// TwinCAT 3 PLC project plc01
// ProgramVersion: 3.1.4026.19
// libraries:
//   Tc2_Standard, * (Beckhoff Automation GmbH)
//   Tc2_System, * (Beckhoff Automation GmbH)
//   Tc2_Utilities, * (Beckhoff Automation GmbH)
//   Tc3_Event, * (www.peterzerlauth.com)
// project tree:
//   / FastTask.TcTTO (not stored), PlcTask.TcTTO (not stored)
//   POUs/ FAST.TcPOU, FB_TestSlow.TcPOU, FB_TestFast.TcPOU, FB_Test1000.TcPOU, MAIN.TcPOU
// real-time tasks:
//   TASK SlowTask: cycle T#20ms, priority 20, ADS port 350
//   TASK FastTask: cycle T#1ms, priority 1, ADS port 351

// ---- POUs/FAST.TcPOU
PROGRAM FAST
VAR
	fbTest:			FB_TestFast;
  	exception:			__SYSTEM.ExceptionCode;	
END_VAR

__TRY
	IF exception = __SYSTEM.ExceptionCode.RTSEXCPT_NOEXCEPTION THEN
// 		fbTest.P_Event.P_Logger:= MAIN.fbLogger;
	
	fbTest();
	
		
	END_IF


__CATCH(exception)


__ENDTRY

END_PROGRAM

// ---- POUs/FB_TestFast.TcPOU
FUNCTION_BLOCK FB_TestFast
VAR_INPUT
END_VAR
VAR_OUTPUT
END_VAR
VAR
	fbEvent: 			Tc3_Event.FB_Event;
	bVerbose:			BOOL;
	bInfo:				BOOL;
	bWarning:			BOOL;
	bError:				BOOL;
	bCritical:			BOOL;

END_VAR

fbEvent();

// Demonstration of FB_Event usage with various log levels and argument types

IF bVerbose THEN
	fbEvent.P_Argument.M_AddINT(134052566194980000);
	fbEvent.P_Argument.M_AddSTRING('mm');
	fbEvent.M_Verbose('V message %s %s');
END_IF

IF bInfo THEN
	fbEvent.P_Argument.M_AddREAL(33.134581234, 3);
	fbEvent.P_Argument.M_AddSTRING('mm');
	fbEvent.M_Info(828536003, 'I message %s %s');
END_IF

IF bWarning THEN
	fbEvent.M_Warning(475719253, 'W message');
	fbEvent.M_Warning(475719253, 'W message');
END_IF

IF bError THEN
	fbEvent.M_Error(475719235, 'E message');
END_IF

IF bCritical THEN
	fbEvent.M_Critical(475719233, 'C message'); ///839384782
END_IF

PROPERTY PUBLIC P_Event : reference to FB_event
GET
P_Event ref= fbEvent;
END_GET
END_PROPERTY

END_FUNCTION_BLOCK

// ---- POUs/FB_TestSlow.TcPOU
FUNCTION_BLOCK FB_TestSlow
VAR_INPUT
END_VAR
VAR_OUTPUT
END_VAR
VAR
	fbEvent: 			Tc3_Event.FB_Event;
	bVerbose:			BOOL;
	bInfo:				BOOL;
	bWarning:			BOOL;
	bError:				BOOL;
	bCritical:			BOOL;

END_VAR

fbEvent();

// Demonstration of FB_Event usage with various log levels and argument types

IF bVerbose THEN
	fbEvent.P_Argument.M_AddINT(134052566194980000);
	fbEvent.P_Argument.M_AddSTRING('mm');
	fbEvent.M_Verbose('V message %s %s');
END_IF

IF bInfo THEN
	fbEvent.P_Argument.M_AddREAL(33.134581234, 3);
	fbEvent.P_Argument.M_AddSTRING('mm');
	fbEvent.M_Info(828536003, 'I message %s %s');
END_IF

IF bWarning THEN
	fbEvent.M_Warning(475719253, 'W message');
	fbEvent.M_Warning(475719253, 'W message');
END_IF

IF bError THEN
	fbEvent.M_Error(475719235, 'E message');
END_IF

IF bCritical THEN
	fbEvent.M_Critical(475719233, 'C message'); ///839384782
	fbEvent.M_Error(849363082, 'Input %s is simulated');
END_IF

PROPERTY PUBLIC P_Event : reference to FB_event
GET
P_Event ref= fbEvent;
END_GET
END_PROPERTY

END_FUNCTION_BLOCK

// ---- POUs/FB_Test1000.TcPOU
FUNCTION_BLOCK FB_Test1000
VAR_INPUT
END_VAR
VAR_OUTPUT
END_VAR
VAR
	fbEvent: 			Tc3_Event.FB_Event;
	bVerbose:			BOOL;
	bInfo:				BOOL;
	bWarning:			BOOL;
	bError:				BOOL;
	bCritical:			BOOL;

END_VAR

fbEvent.M_Error(767040015, 'Failed to load recipe: %s');
fbEvent.M_Error(945171139, 'Gate interlock failed');
fbEvent.M_Error(672737192, 'Proximity sensor %s is faulty');
fbEvent.M_Error(218555824, 'System voltage is unstable');
fbEvent.M_Error(378958620, 'Data packet from robot is corrupt');
fbEvent.M_Error(100559308, 'Cylinder B did not retract within timeout');
fbEvent.M_Error(422522142, 'Main drive overtemperature');
fbEvent.M_Error(109177156, 'Network switch communication error');
fbEvent.M_Error(728320830, 'Operator login failed for user %s');
fbEvent.M_Error(842704677, 'Tool change failed on station %s');
fbEvent.M_Error(114606201, 'Regulator pressure is out of range');
fbEvent.M_Error(69032799, 'Homing failed for axis %s');
fbEvent.M_Error(6079279, 'Chiller fluid level is low');
fbEvent.M_Error(403905948, 'Vision system could not locate part %s');
fbEvent.M_Error(572693817, 'Fire suppression system activated');
fbEvent.M_Error(493750134, 'Motor B thermal overload');
fbEvent.M_Error(185108713, 'Analog input %s signal out of range');
fbEvent.M_Error(650556097, 'Palletizer stack height error');
fbEvent.M_Error(361596979, 'Failed to write to database');
fbEvent.M_Error(927599790, 'Inconsistent barcode scan for part %s');
fbEvent.M_Error(445448130, 'Axis %s software limit switch triggered');
fbEvent.M_Error(516547226, 'Manual mode interlock is active');
fbEvent.M_Error(461325003, 'Leak detected in hydraulic line %s');
fbEvent.M_Error(213620218, 'Pressure relief valve is active');
fbEvent.M_Error(970539493, 'PLC CPU temperature is high');
fbEvent.M_Error(250388329, 'Cannot open file %s on HMI');
fbEvent.M_Error(777930705, 'Watchdog timer has expired');
fbEvent.M_Error(801846437, 'Clamping force not achieved');
fbEvent.M_Error(96634275, 'Emergency stop chain is broken');
fbEvent.M_Error(737238189, 'Proximity sensor 4 did not detect part');
fbEvent.M_Error(306046057, 'Axis 2 position deviation too high');
fbEvent.M_Error(224203696, 'Communication with VFD %s failed');
fbEvent.M_Error(157553850, 'Air filter is clogged');
fbEvent.M_Error(138291755, 'Incorrect part orientation detected');
fbEvent.M_Error(147243850, 'System failed to initialize');
fbEvent.M_Error(674332993, 'Torque limit exceeded for motor %s');
fbEvent.M_Error(892736622, 'Sensor supply voltage is low');
fbEvent.M_Error(233128167, 'Safety relay test failed');
fbEvent.M_Error(189564922, 'Cycle start not permitted: Guard open');
fbEvent.M_Error(133354980, 'Invalid command received from HMI');
fbEvent.M_Error(474590038, 'Conveyor speed is below setpoint');
fbEvent.M_Error(111102940, 'Failed to grip part at station %s');
fbEvent.M_Error(454980182, 'Hydraulic fluid level is critically low');
fbEvent.M_Error(21914838, 'Temperature sensor %s is disconnected');
fbEvent.M_Error(459705985, 'Robot is in singularity position');
fbEvent.M_Error(643839111, 'Network connection to SCADA lost');
fbEvent.M_Error(152217629, 'Axis %s hardware limit switch triggered');
fbEvent.M_Error(53648101, 'Pump motor failed to start');
fbEvent.M_Error(825497978, 'Mode change failed: System not in safe state');
fbEvent.M_Error(650351655, 'Error in motion group %s');
fbEvent.M_Error(570390914, 'Lubrication system fault');
fbEvent.M_Error(395794439, 'Failed to close valve %s');
fbEvent.M_Error(668897735, 'Excessive vibration detected on motor %s');
fbEvent.M_Error(183659276, 'Part presence sensor stuck on');
fbEvent.M_Error(831292259, 'Batch number %s is invalid or expired');
fbEvent.M_Error(334820327, 'Main circuit breaker is tripped');
fbEvent.M_Error(817895218, 'Failed to establish connection to robot %s');
fbEvent.M_Error(829414129, 'Pressure sensor reading is frozen');
fbEvent.M_Error(699628057, 'Cylinder A extended unexpectedly');
fbEvent.M_Error(586587708, 'Insufficient air pressure for gripper');
fbEvent.M_Error(389909287, 'E-Stop reset failed: Fault condition still present');
fbEvent.M_Error(574025698, 'Encoder battery voltage is low');
fbEvent.M_Error(124048137, 'Invalid parameter set for drive %s');
fbEvent.M_Error(503377368, 'Flow rate is too low in line %s');
fbEvent.M_Error(727034518, 'Homing sequence interrupted');
fbEvent.M_Error(997482720, 'Safety mat is active');
fbEvent.M_Error(245800601, 'PLC scan time is too high');
fbEvent.M_Error(21062406, 'Configuration file %s is corrupted');
fbEvent.M_Error(190843921, 'Axis %s stalled during movement');
fbEvent.M_Error(703927388, 'Temperature out of spec for oven %s');
fbEvent.M_Error(58246198, 'Failed to eject part from mold');
fbEvent.M_Error(167321371, 'Wrong tool loaded in spindle');
fbEvent.M_Error(912727106, 'Robot path planning error for destination %s');
fbEvent.M_Error(103282373, 'Overvoltage detected on DC bus');
fbEvent.M_Error(833526939, 'Purge cycle failed to complete');
fbEvent.M_Error(271146146, 'Signal conflict between two sensors');
fbEvent.M_Error(739531565, 'Cannot load G-code file: %s');
fbEvent.M_Error(691039117, 'Failed to enable drive group %s');
fbEvent.M_Error(580723245, 'Reservoir level is high');
fbEvent.M_Error(187382456, 'Welding tip is worn');
fbEvent.M_Error(513756036, 'Incorrect fixture ID %s received');
fbEvent.M_Error(197253253, 'Servo motor overheating');
fbEvent.M_Error(186009301, 'Failed to close safety gate');
fbEvent.M_Error(459468574, 'Sensor fault: Short circuit');
fbEvent.M_Error(450883362, 'PLC memory is full');
fbEvent.M_Error(617100714, 'Actuator %s did not complete motion');
fbEvent.M_Error(681586278, 'Part quality check failed at station %s');
fbEvent.M_Error(250193368, 'Main contactor did not engage');
fbEvent.M_Error(585312983, 'System is in E-Stop state');
fbEvent.M_Error(248322796, 'Analog output %s is at fault');
fbEvent.M_Error(907814064, 'Failed to read data from RFID tag');
fbEvent.M_Error(909421439, 'Conveyor index timeout');
fbEvent.M_Error(973163742, 'Emergency stop line is broken');
fbEvent.M_Error(976950794, 'Axis %s is not referenced');
fbEvent.M_Error(96700224, 'Valve manifold communication error');
fbEvent.M_Error(325249016, 'Temperature ramp rate too fast');
fbEvent.M_Error(16987038, 'Failed to synchronize axes');
fbEvent.M_Error(902100387, 'Robot joint %s limit exceeded');
fbEvent.M_Error(47762990, 'Vision system lighting failure');
fbEvent.M_Error(895266560, 'Pressure sensor %s shows maximum value');
fbEvent.M_Error(458251234, 'Machine not homed');
fbEvent.M_Error(920133186, 'User %s does not have required permissions');
fbEvent.M_Error(211254420, 'Hydraulic accumulator is pre-charged incorrectly');
fbEvent.M_Error(358912044, 'Coolant flow switch is open');
fbEvent.M_Error(163821495, 'Part jam detected in chute %s');
fbEvent.M_Error(719723582, 'Failed to zero axis %s');
fbEvent.M_Error(518915054, 'Motor phase loss detected');
fbEvent.M_Error(107984654, 'Internal PLC error: Task overrun');
fbEvent.M_Error(394586519, 'Barcode scanner not ready');
fbEvent.M_Error(466512842, 'Invalid move command for axis %s');
fbEvent.M_Error(920835287, 'Safety PLC communication fault');
fbEvent.M_Error(877440804, 'Filter differential pressure is high');
fbEvent.M_Error(650467130, 'Cylinder B pressure not building');
fbEvent.M_Error(483921545, 'Spindle speed not reached');
fbEvent.M_Error(518106258, 'Robot collision detected');
fbEvent.M_Error(694145951, 'Failed to update recipe %s in database');
fbEvent.M_Error(324626171, 'Interlock condition not met for operation %s');
fbEvent.M_Error(276535387, 'System pressure is too high');
fbEvent.M_Error(100381264, 'VFD in fault state');
fbEvent.M_Error(201466115, 'HMI backup failed');
fbEvent.M_Error(646466444, 'Position feedback lost for axis %s');
fbEvent.M_Error(833582598, 'Label printer error: Out of labels');
fbEvent.M_Error(642342615, 'Chiller temperature is too high');
fbEvent.M_Error(853428607, 'Part unloading failed');
fbEvent.M_Error(493067428, 'Emergency stop reset timeout');
fbEvent.M_Error(82768936, 'Axis %s command position and actual position mismatch');
fbEvent.M_Error(169365827, 'Pump is running dry');
fbEvent.M_Error(775018957, 'Level sensor in tank %s is faulted');
fbEvent.M_Error(395644558, 'Failed to park robot');
fbEvent.M_Error(876255699, 'Conveyor motor overload');
fbEvent.M_Error(722100646, 'Wrong material loaded for job %s');
fbEvent.M_Error(755117431, 'Air compressor fault');
fbEvent.M_Error(558772479, 'PLC I/O module error');
fbEvent.M_Error(10818780, 'Excessive cycle time detected');
fbEvent.M_Error(622567336, 'Safety gate switch is welded');
fbEvent.M_Error(171563348, 'Failed to open valve %s');
fbEvent.M_Error(738933589, 'Thermocouple %s is broken');
fbEvent.M_Error(946961693, 'Cylinder A failed to extend');
fbEvent.M_Error(241776719, 'Robot is not in auto mode');
fbEvent.M_Error(989752245, 'System failed to shutdown gracefully');
fbEvent.M_Error(995549063, 'Load cell signal is unstable');
fbEvent.M_Error(598954565, 'Homing timeout for axis %s');
fbEvent.M_Error(368168081, 'Purge valve is stuck open');
fbEvent.M_Error(918018155, 'Network cable unplugged for device %s');
fbEvent.M_Error(632543431, 'Operator intervention required');
fbEvent.M_Error(875369228, 'Failed to apply torque on fastener %s');
fbEvent.M_Error(278050376, 'Proximity sensor fault: Wire break');
fbEvent.M_Error(976000847, 'Main power supply failure');
fbEvent.M_Error(478766911, 'Robot program %s is not found');
fbEvent.M_Error(240496535, 'VFD overcurrent trip');
fbEvent.M_Error(796761515, 'Cylinder B failed to retract');
fbEvent.M_Error(887975720, 'Failed to maintain pressure at %s bar');
fbEvent.M_Error(730300082, 'Axis %s brake did not release');
fbEvent.M_Error(873262718, 'HMI screen saver is active');
fbEvent.M_Error(461991977, 'Failed to enable safety outputs');
fbEvent.M_Error(850383252, 'Part transfer failed');
fbEvent.M_Error(130699376, 'Incorrect password entered %s times');
fbEvent.M_Error(787416019, 'Sensor %s is dirty or misaligned');
fbEvent.M_Error(923173815, 'Spindle tool not clamped');
fbEvent.M_Error(268499768, 'System is in maintenance mode');
fbEvent.M_Error(593854326, 'Failed to log data to file %s');
fbEvent.M_Error(450978005, 'Conveyor belt slipped');
fbEvent.M_Error(189339750, 'Hydraulic fluid is contaminated');
fbEvent.M_Error(632933750, 'Robot joint %s temperature is high');
fbEvent.M_Error(817837904, 'Axis 3 move command cancelled');
fbEvent.M_Error(624086393, 'Light curtain fault: Mutingshort circuit');
fbEvent.M_Error(56417063, 'PLC battery needs replacement');
fbEvent.M_Error(26494080, 'Failed to connect to MES system');
fbEvent.M_Error(307474215, 'Weight of part %s is out of tolerance');
fbEvent.M_Error(539723334, 'Air dryer fault');
fbEvent.M_Error(770448370, 'Valve %s did not shift');
fbEvent.M_Error(524419490, 'Safety relay did not pick up');
fbEvent.M_Error(335177129, 'Failed to find reference mark for axis %s');
fbEvent.M_Error(308668500, 'Temperature in zone %s is too low');
fbEvent.M_Error(722667901, 'Clamp pressure not released');
fbEvent.M_Error(696415796, 'Robot path obstructed');
fbEvent.M_Error(247141302, 'Failed to save settings to HMI');
fbEvent.M_Error(901105930, 'Motor B is not responding');
fbEvent.M_Error(819946865, 'Proximity sensor %s is always on');
fbEvent.M_Error(284135205, 'System pressure not building');
fbEvent.M_Error(130581478, 'Failed to execute command %s');
fbEvent.M_Error(374393878, 'E-Stop source: Panel Button');
fbEvent.M_Error(322717611, 'Axis %s is disabled');
fbEvent.M_Error(401150847, 'Pump suction is clogged');
fbEvent.M_Error(733087097, 'Failed to read configuration from drive');
fbEvent.M_Error(216165052, 'Part height is incorrect at station %s');
fbEvent.M_Error(443472917, 'Robot is in singularity, cannot move');
fbEvent.M_Error(667295922, 'VFD undervoltage fault');
fbEvent.M_Error(954889344, 'Cylinder A pressure sensor fault');
fbEvent.M_Error(801470049, 'Safety gate not locked');
fbEvent.M_Error(354268224, 'Failed to write to I/O module %s');
fbEvent.M_Error(814712779, 'Encoder resolution mismatch');
fbEvent.M_Error(15257384, 'Spindle speed is zero');
fbEvent.M_Error(507544693, 'System failed to enter run mode');
fbEvent.M_Error(400693354, 'Pallet not present at location %s');
fbEvent.M_Error(449222015, 'Hydraulic return filter is clogged');
fbEvent.M_Error(567617912, 'Robot gripper failed to open');
fbEvent.M_Error(805648219, 'PLC time sync failed');
fbEvent.M_Error(61520055, 'Failed to find part %s in vision system');
fbEvent.M_Error(673927967, 'Conveyor tracking lost');
fbEvent.M_Error(131126122, 'Emergency stop source: Pull Cord');
fbEvent.M_Error(91674575, 'Axis %s brake did not engage');
fbEvent.M_Error(165763222, 'Motor A thermal model trip');
fbEvent.M_Error(599082815, 'Level sensor in tank %s is frozen');
fbEvent.M_Error(580024245, 'Failed to close gripper');
fbEvent.M_Error(809869490, 'Safety light curtain is muted');
fbEvent.M_Error(990910834, 'VFD DC bus overvoltage');
fbEvent.M_Error(815430670, 'Cylinder B extended unexpectedly');
fbEvent.M_Error(894832746, 'Failed to start cycle: Guard not closed');
fbEvent.M_Error(617683718, 'Robot is in manual mode');
fbEvent.M_Error(315414856, 'System pressure relief valve active');
fbEvent.M_Error(413433193, 'Failed to load G-code: Invalid syntax');
fbEvent.M_Error(591728841, 'Axis %s is not homed');
fbEvent.M_Error(417679101, 'Motor C bearing failure');
fbEvent.M_Error(193631627, 'Air pressure is too high');
fbEvent.M_Error(662248344, 'Failed to park robot in home position');
fbEvent.M_Error(853313589, 'HMI firmware update failed');
fbEvent.M_Error(434502460, 'E-Stop source: Gateway');
fbEvent.M_Error(814923249, 'Proximity sensor %s is always off');
fbEvent.M_Error(794917286, 'Temperature ramp rate too slow');
fbEvent.M_Error(581947941, 'Failed to open gripper');
fbEvent.M_Error(31918372, 'Robot collision detected at joint %s');
fbEvent.M_Error(50407106, 'VFD motor stall');
fbEvent.M_Error(680958902, 'Cylinder A failed to retract');
fbEvent.M_Error(895803704, 'Failed to maintain speed at %s RPM');
fbEvent.M_Error(572177518, 'Safety PLC test failed');
fbEvent.M_Error(245219383, 'Failed to read barcode from part %s');
fbEvent.M_Error(264827515, 'Conveyor motor is not running');
fbEvent.M_Error(516448418, 'Emergency stop source: Safety Mat');
fbEvent.M_Error(903016714, 'Axis %s is in alarm state');
fbEvent.M_Error(624130335, 'Pump discharge is blocked');
fbEvent.M_Error(15017611, 'Failed to execute robot program %s');
fbEvent.M_Error(312928369, 'System is in E-Stop state: Reset required');
fbEvent.M_Error(807217067, 'Motor D overtemperature');
fbEvent.M_Error(707206051, 'Air leak detected in circuit %s');
fbEvent.M_Error(362431411, 'Failed to close valve manifold');
fbEvent.M_Error(883541551, 'Safety gate not closed');
fbEvent.M_Error(603033245, 'Failed to set output %s');
fbEvent.M_Error(586589094, 'Encoder count error');
fbEvent.M_Error(187121568, 'Spindle direction is incorrect');
fbEvent.M_Error(108014721, 'System failed to initialize I/O');
fbEvent.M_Error(136578612, 'Pallet is skewed at location %s');
fbEvent.M_Error(984349400, 'Hydraulic pump is noisy');
fbEvent.M_Error(151356623, 'Robot gripper failed to close');
fbEvent.M_Error(249651244, 'PLC network redundancy lost');
fbEvent.M_Error(999593972, 'Failed to find fiducial %s in vision system');
fbEvent.M_Error(506729989, 'Conveyor belt is torn');
fbEvent.M_Error(967408081, 'Emergency stop source: Dual Channel');
fbEvent.M_Error(91123471, 'Axis %s following error is active');
fbEvent.M_Error(700443361, 'Motor E bearing temperature is high');
fbEvent.M_Error(447311786, 'Air pressure is too low');
fbEvent.M_Error(635308455, 'Failed to move robot to safe position');
fbEvent.M_Error(87546593, 'HMI application crashed');
fbEvent.M_Error(554740636, 'E-Stop source: Hardwired');
fbEvent.M_Error(925410774, 'Proximity sensor %s is intermittent');
fbEvent.M_Error(390584469, 'Temperature overshoot detected');
fbEvent.M_Error(830463546, 'Failed to release part');
fbEvent.M_Error(809577234, 'Robot joint limit reached');
fbEvent.M_Error(647484742, 'VFD motor overload');
fbEvent.M_Error(699628057, 'Cylinder A extended unexpectedly');
fbEvent.M_Error(896554714, 'Failed to maintain torque at %s Nm');
fbEvent.M_Error(340736568, 'Safety relay test passed with warnings');
fbEvent.M_Error(424019756, 'Failed to write barcode to part %s');
fbEvent.M_Error(759279025, 'Conveyor speed is zero');
fbEvent.M_Error(224304038, 'Emergency stop source: Unlisted');
fbEvent.M_Error(488694884, 'Axis %s is not enabled');
fbEvent.M_Error(13330519, 'Pump cavitation detected');
fbEvent.M_Error(511958330, 'Failed to load robot program %s');
fbEvent.M_Error(5835009, 'System is in fault state: Reset required');
fbEvent.M_Error(632413153, 'Motor F overcurrent');
fbEvent.M_Error(177442738, 'Air dryer is saturated');
fbEvent.M_Error(418168403, 'Failed to open safety valve');
fbEvent.M_Error(921825778, 'Safety gate is not interlocked');
fbEvent.M_Error(892005793, 'Failed to clear output %s');
fbEvent.M_Error(540454385, 'Encoder signal is noisy');
fbEvent.M_Error(52190518, 'Spindle tool is broken');
fbEvent.M_Error(147858480, 'System failed to load configuration');
fbEvent.M_Error(55697345, 'Pallet is missing at location %s');
fbEvent.M_Error(382288216, 'Hydraulic fluid is low');
fbEvent.M_Error(333901242, 'Robot gripper is worn');
fbEvent.M_Error(262534927, 'PLC task watchdog has expired');
fbEvent.M_Error(198734585, 'Failed to match pattern %s in vision system');
fbEvent.M_Error(391356591, 'Conveyor motor is overheating');
fbEvent.M_Error(153010784, 'Emergency stop source: Software');
fbEvent.M_Error(705339355, 'Axis %s is in warning state');
fbEvent.M_Error(106531401, 'Motor G is not calibrated');
fbEvent.M_Error(908161022, 'Air pressure is unstable');
fbEvent.M_Error(242227519, 'Failed to power down robot');
fbEvent.M_Error(14472554, 'HMI display is faulty');
fbEvent.M_Error(249490462, 'E-Stop source: External');
fbEvent.M_Error(605066668, 'Proximity sensor %s is miswired');
fbEvent.M_Error(886870306, 'Temperature undershoot detected');
fbEvent.M_Error(926405723, 'Failed to grip part');
fbEvent.M_Error(12352681, 'Robot software limit reached');
fbEvent.M_Error(814091696, 'VFD communication is lost');
fbEvent.M_Error(62764297, 'Cylinder B failed to extend');
fbEvent.M_Error(817611067, 'Failed to maintain position at %s mm');
fbEvent.M_Error(601814376, 'Safety relay test failed critically');
fbEvent.M_Error(461206374, 'Failed to verify barcode on part %s');
fbEvent.M_Error(319540893, 'Conveyor is overloaded');
fbEvent.M_Error(213764771, 'Emergency stop source: Unknown');
fbEvent.M_Error(990418917, 'Axis %s is in fault state');
fbEvent.M_Error(108261308, 'Pump efficiency is low');
fbEvent.M_Error(514776885, 'Failed to save robot program %s');
fbEvent.M_Error(384404749, 'System is in safe state');
fbEvent.M_Error(997626545, 'Motor H has a ground fault');
fbEvent.M_Error(92074348, 'Air filter is dirty');
fbEvent.M_Error(402112666, 'Failed to close isolation valve');
fbEvent.M_Error(138780411, 'Safety gate is open');
fbEvent.M_Error(754317046, 'Failed to set input %s');
fbEvent.M_Error(810684995, 'Encoder battery is dead');
fbEvent.M_Error(235849703, 'Spindle is not running');
fbEvent.M_Error(257990122, 'System failed to boot');
fbEvent.M_Error(152167975, 'Pallet is double-stacked at location %s');
fbEvent.M_Error(171706880, 'Hydraulic fluid is overheating');
fbEvent.M_Error(292450194, 'Robot gripper is damaged');
fbEvent.M_Error(822620336, 'PLC scan time is too long');
fbEvent.M_Error(472161434, 'Failed to locate feature %s in vision system');
fbEvent.M_Error(867753627, 'Conveyor belt is misaligned');
fbEvent.M_Error(435208140, 'Emergency stop has been reset');
fbEvent.M_Error(517173547, 'Axis %s is homed');
fbEvent.M_Error(995328853, 'Motor I is not configured');
fbEvent.M_Error(107546264, 'Air pressure is normal');
fbEvent.M_Error(45270352, 'Failed to power on robot');
fbEvent.M_Error(704170036, 'HMI is connected');
fbEvent.M_Error(922682629, 'E-Stop source is clear');
fbEvent.M_Error(879160142, 'Proximity sensor %s is working');
fbEvent.M_Error(518169734, 'Temperature is stable');
fbEvent.M_Error(446837303, 'Part is gripped');
fbEvent.M_Error(947331221, 'Robot is in home position');
fbEvent.M_Error(101908288, 'VFD is running');
fbEvent.M_Error(555525126, 'Cylinder A is retracted');
fbEvent.M_Error(897554373, 'Position is correct at %s mm');
fbEvent.M_Error(260834187, 'Safety system is OK');
fbEvent.M_Error(826896815, 'Barcode on part %s is verified');
fbEvent.M_Error(50359082, 'Conveyor is running');
fbEvent.M_Error(740668744, 'System is in run mode');
fbEvent.M_Error(406934296, 'Axis %s is enabled');
fbEvent.M_Error(146319251, 'Pump is running');
fbEvent.M_Error(276082621, 'Robot program %s is loaded');
fbEvent.M_Error(108094323, 'System is ready');
fbEvent.M_Error(230514679, 'Motor J is OK');
fbEvent.M_Error(832896431, 'Air system is OK');
fbEvent.M_Error(656692625, 'Valve is open');
fbEvent.M_Error(715667115, 'Safety gate is closed and locked');
fbEvent.M_Error(466230381, 'Input %s is on');
fbEvent.M_Error(788683792, 'Encoder is working');
fbEvent.M_Error(738571353, 'Spindle is at speed');
fbEvent.M_Error(453904248, 'System is booted');
fbEvent.M_Error(850980581, 'Pallet is at location %s');
fbEvent.M_Error(71608016, 'Hydraulic system is OK');
fbEvent.M_Error(725313717, 'Robot gripper is open');
fbEvent.M_Error(383890713, 'PLC is running');
fbEvent.M_Error(494356061, 'Vision system is ready');
fbEvent.M_Error(111775791, 'Conveyor is stopped');
fbEvent.M_Error(512901664, 'System is in auto mode');
fbEvent.M_Error(466641342, 'Axis %s is stopped');
fbEvent.M_Error(815156172, 'Pump is stopped');
fbEvent.M_Error(514934417, 'Robot is idle');
fbEvent.M_Error(164924335, 'System is in manual mode');
fbEvent.M_Error(144721828, 'Motor K is stopped');
fbEvent.M_Error(311040202, 'Air system is off');
fbEvent.M_Error(265293020, 'Valve is closed');
fbEvent.M_Error(854716410, 'Safety gate is unlocked');
fbEvent.M_Error(650944564, 'Input %s is off');
fbEvent.M_Error(564745397, 'Encoder is not connected');
fbEvent.M_Error(538297842, 'Spindle is stopped');
fbEvent.M_Error(653475126, 'System is shutting down');
fbEvent.M_Error(13621109, 'Pallet is empty at location %s');
fbEvent.M_Error(675619028, 'Hydraulic system is off');
fbEvent.M_Error(477738670, 'Robot gripper is closed');
fbEvent.M_Error(347913332, 'PLC is stopped');
fbEvent.M_Error(940536226, 'Vision system is off');
fbEvent.M_Error(664414487, 'Conveyor is jammed');
fbEvent.M_Error(298911306, 'System is in fault');
fbEvent.M_Error(305930856, 'Axis %s is moving');
fbEvent.M_Error(105663102, 'Pump is priming');
fbEvent.M_Error(180650545, 'Robot is moving');
fbEvent.M_Error(336903017, 'System is initializing');
fbEvent.M_Error(143184871, 'Motor L is starting');
fbEvent.M_Error(133408958, 'Air system is charging');
fbEvent.M_Error(53324685, 'Valve is shifting');
fbEvent.M_Error(671524722, 'Safety gate is opening');
fbEvent.M_Error(636838680, 'Input %s is faulted');
fbEvent.M_Error(809572133, 'Encoder is homing');
fbEvent.M_Error(337441676, 'Spindle is starting');
fbEvent.M_Error(830120866, 'System is saving data');
fbEvent.M_Error(766296111, 'Pallet is arriving at location %s');
fbEvent.M_Error(983074762, 'Hydraulic system is charging');
fbEvent.M_Error(99444800, 'Robot gripper is releasing');
fbEvent.M_Error(732461370, 'PLC is in program mode');
fbEvent.M_Error(240623418, 'Vision system is capturing image');
fbEvent.M_Error(499405395, 'Conveyor is indexing');
fbEvent.M_Error(255896736, 'System is in config mode');
fbEvent.M_Error(270934408, 'Axis %s is referencing');
fbEvent.M_Error(801929015, 'Pump is building pressure');
fbEvent.M_Error(115614024, 'Robot is referencing');
fbEvent.M_Error(598382864, 'System is in test mode');
fbEvent.M_Error(947105744, 'Motor M is running');
fbEvent.M_Error(758812146, 'Air system is at pressure');
fbEvent.M_Error(680818073, 'Valve is energized');
fbEvent.M_Error(538649955, 'Safety gate is closing');
fbEvent.M_Error(653377590, 'Input %s is simulated');
fbEvent.M_Error(902808007, 'Encoder is synchronized');
fbEvent.M_Error(512875126, 'Spindle is braking');
fbEvent.M_Error(70786942, 'System is online');
fbEvent.M_Error(959258201, 'Pallet is leaving location %s');
fbEvent.M_Error(725485121, 'Hydraulic system is active');
fbEvent.M_Error(282561217, 'Robot gripper is gripping');
fbEvent.M_Error(960505020, 'PLC is in run mode');
fbEvent.M_Error(955690866, 'Vision system is processing image');
fbEvent.M_Error(615290565, 'Conveyor is accelerating');
fbEvent.M_Error(414835851, 'System is in service mode');
fbEvent.M_Error(914575188, 'Axis %s is waiting');
fbEvent.M_Error(770266437, 'Pump is at speed');
fbEvent.M_Error(685129588, 'Robot is waiting for input');
fbEvent.M_Error(11345948, 'System is in standby');
fbEvent.M_Error(637572567, 'Motor N is at temperature');
fbEvent.M_Error(106218867, 'Air system is venting');
fbEvent.M_Error(97019314, 'Valve is de-energized');
fbEvent.M_Error(424182736, 'Safety gate is locked');
fbEvent.M_Error(368754980, 'Input %s is forced');
fbEvent.M_Error(264421939, 'Encoder is at zero');
fbEvent.M_Error(220452105, 'Spindle is changing tool');
fbEvent.M_Error(47796760, 'System is offline');
fbEvent.M_Error(955956074, 'Pallet is at position %s');
fbEvent.M_Error(380578516, 'Hydraulic system is idle');
fbEvent.M_Error(174104869, 'Robot gripper is empty');
fbEvent.M_Error(717293661, 'PLC is in fault mode');
fbEvent.M_Error(539938012, 'Vision system failed to focus');
fbEvent.M_Error(342459851, 'Conveyor is decelerating');
fbEvent.M_Error(636971575, 'System is in emergency stop');
fbEvent.M_Error(67668378, 'Axis %s is in error');
fbEvent.M_Error(510870299, 'Pump is in alarm');
fbEvent.M_Error(835699300, 'Robot is in error');
fbEvent.M_Error(646261057, 'System is in safe stop');
fbEvent.M_Error(949812312, 'Motor O is in alarm');
fbEvent.M_Error(20308516, 'Air system is in fault');
fbEvent.M_Error(992338084, 'Valve is in fault');
fbEvent.M_Error(605437452, 'Safety gate is in fault');
fbEvent.M_Error(298543865, 'Input %s is in error');
fbEvent.M_Error(298239697, 'Encoder is in alarm');
fbEvent.M_Error(633513693, 'Spindle is in fault');
fbEvent.M_Error(230331814, 'System is in power save');
fbEvent.M_Error(984735048, 'Pallet is damaged at location %s');
fbEvent.M_Error(685765076, 'Hydraulic system is in fault');
fbEvent.M_Error(578797095, 'Robot gripper is in fault');
fbEvent.M_Error(71142695, 'PLC is in stop mode');
fbEvent.M_Error(242242005, 'Vision system is in error');
fbEvent.M_Error(17659654, 'Conveyor is in E-Stop');
fbEvent.M_Error(939635885, 'System is in maintenance');
fbEvent.M_Error(322717611, 'Axis %s is disabled');
fbEvent.M_Error(799635987, 'Pump is disabled');
fbEvent.M_Error(150713939, 'Robot is disabled');
fbEvent.M_Error(751474474, 'System is in setup');
fbEvent.M_Error(997394142, 'Motor P is disabled');
fbEvent.M_Error(883170496, 'Air system is disabled');
fbEvent.M_Error(170395681, 'Valve is disabled');
fbEvent.M_Error(531330424, 'Safety gate is disabled');
fbEvent.M_Error(735365405, 'Input %s is disabled');
fbEvent.M_Error(146502318, 'Encoder is disabled');
fbEvent.M_Error(394374111, 'Spindle is disabled');
fbEvent.M_Error(688320457, 'System is in reset');
fbEvent.M_Error(165346795, 'Pallet is missing from location %s');
fbEvent.M_Error(168985146, 'Hydraulic system is disabled');
fbEvent.M_Error(126276672, 'Robot gripper is disabled');
fbEvent.M_Error(90348213, 'PLC is in reset');
fbEvent.M_Error(56057379, 'Vision system is disabled');
fbEvent.M_Error(735885173, 'Conveyor is in reset');
fbEvent.M_Error(376915595, 'System is in power up');
fbEvent.M_Error(509889079, 'Axis %s is powering up');
fbEvent.M_Error(901588235, 'Pump is powering up');
fbEvent.M_Error(922947088, 'Robot is powering up');
fbEvent.M_Error(178852797, 'System is in power down');
fbEvent.M_Error(55561347, 'Motor Q is powering down');
fbEvent.M_Error(111232102, 'Air system is powering down');
fbEvent.M_Error(396735236, 'Valve is powering down');
fbEvent.M_Error(969610107, 'Safety gate is powering down');
fbEvent.M_Error(512741635, 'Input %s is powering down');
fbEvent.M_Error(5350323, 'Encoder is powering down');
fbEvent.M_Error(253222116, 'Spindle is powering down');
fbEvent.M_Error(624806893, 'System is in communication fault');
fbEvent.M_Error(429580340, 'Pallet is wrong at location %s');
fbEvent.M_Error(481638973, 'Hydraulic system is in communication fault');
fbEvent.M_Error(408793261, 'Robot gripper is in communication fault');
fbEvent.M_Error(91867106, 'PLC is in communication fault');
fbEvent.M_Error(338573968, 'Vision system is in communication fault');
fbEvent.M_Error(785816840, 'Conveyor is in communication fault');
fbEvent.M_Error(507302984, 'System is in configuration fault');
fbEvent.M_Error(272349207, 'Axis %s is in configuration fault');
fbEvent.M_Error(731425804, 'Pump is in configuration fault');
fbEvent.M_Error(626937195, 'Robot is in configuration fault');
fbEvent.M_Error(4807251, 'System is in hardware fault');
fbEvent.M_Error(753322197, 'Motor R is in hardware fault');
fbEvent.M_Error(675446452, 'Air system is in hardware fault');
fbEvent.M_Error(308713644, 'Valve is in hardware fault');
fbEvent.M_Error(845540868, 'Safety gate is in hardware fault');
fbEvent.M_Error(955082190, 'Input %s is in hardware fault');
fbEvent.M_Error(503791964, 'Encoder is in hardware fault');
fbEvent.M_Error(527358624, 'Lag error');
fbEvent.M_Error(467874328, 'Lag error 2');
fbEvent.M_Error(467874328, 'Lag error 3');

PROPERTY PUBLIC P_Event : reference to FB_event
GET
P_Event ref= fbEvent;
END_GET
END_PROPERTY

END_FUNCTION_BLOCK

// ---- POUs/MAIN.TcPOU
PROGRAM MAIN
VAR
	fbLogger:			Tc3_Event.FB_LoggerManager;
	fbHmiLogger:		Tc3_Event.FB_HmiLogger;
	fbFileLogger:		Tc3_Event.FB_FileLogger;
	fbTest:				FB_TestSlow;
	fbTest1000:			FB_Test1000;
  	exception:			__SYSTEM.ExceptionCode;	
	bReset: BOOL;
END_VAR

__TRY
	IF exception = __SYSTEM.ExceptionCode.RTSEXCPT_NOEXCEPTION THEN
		fbLogger.M_Add(fbHmiLogger);
		fbLogger.M_Add(fbFileLogger);
			
		fbHmiLogger();
		fbFileLogger.sPathName:= 'C:\temp\log.txt';
		fbFileLogger();

		
		
		IF bReset THEN
			fbTest.P_Event.M_Reset();
		END_IF
		
		fbTest.P_Event.P_Logger:= fbLogger;
		
		fbTest();	
		
// 		fbTest1000.P_Event.P_Logger:= fbLogger;
// 		fbTest1000();
		
	END_IF

__CATCH(exception)

__ENDTRY

END_PROGRAM
